Omron CX-Programmer project NewProject (CX-Programmer 9.54)

# PLC Station1: CJ1M CPU11

## Global symbols (name address type ; comment)
0.00 BOOL  ; Start_PB
0.01 BOOL  ; Stop_PB
0.02 BOOL  ; Reset_PB
0.03 BOOL  ; Emergency_PB
0.04 BOOL  ; Pusher 1 Front Limit
0.05 BOOL  ; RM Vision
0.06 BOOL  ; Diff_Sensor1
1.00 BOOL  ; RM Emitter
1.01 BOOL  ; Start_Light
1.02 BOOL  ; Stop_Light
1.03 BOOL  ; Reset_Light
1.04 BOOL  ; Pusher 1
1.05 BOOL  ; RM Roller Stopper
1.06 BOOL  ; RM Conveyor
1.07 BOOL  ; Curved RM Conveyor
1.08 BOOL  ; Check RM Conveyor
1.09 BOOL  ; Curved Reject Conveyor
1.10 BOOL  ; Reject RM Conveyor
1.11 BOOL  ; Base Machining Conveyor
D10 CHANNEL  ; Raw Metal Counting
D11 CHANNEL  ; Reject Counting
W10.00 BOOL  ; Pusher_Control
W10.01 BOOL  ; RM Roller Stopper Control
W10.02 BOOL  ; Emitter Control
W10.03 BOOL  ; Reset Counting
W1.00 BOOL  ; Status
W1.01 BOOL  ; Emergency_Status

## Program NewProgram1 (cyclic task 0)

### Section Station1

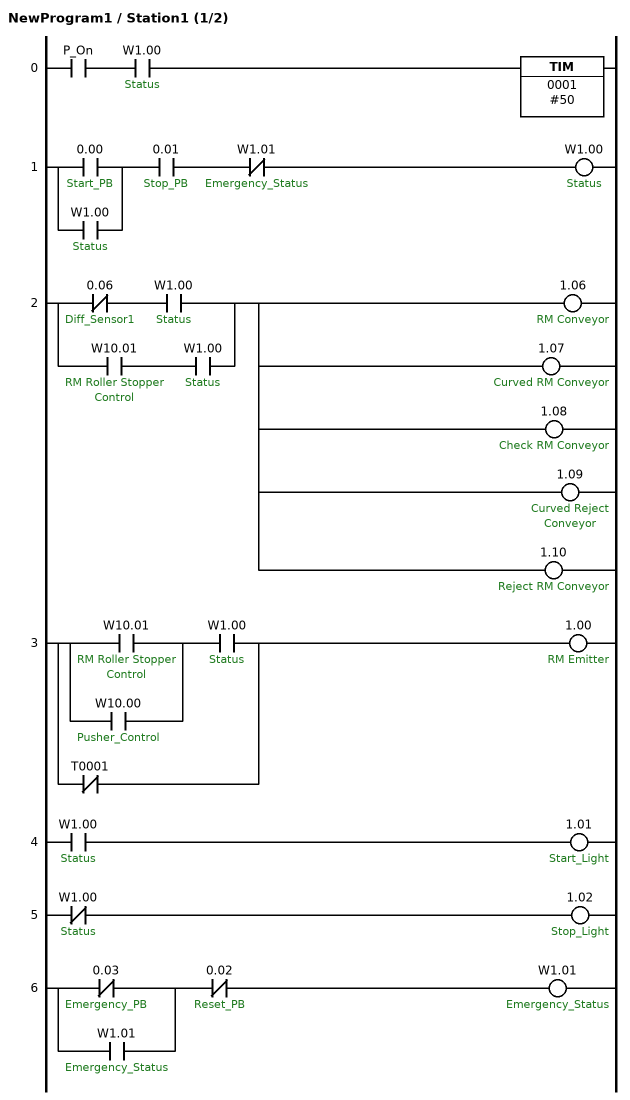
; rung 0
LD P_On
AND W1.00  ; Status
TIM 0001 #50
; rung 1
LD 0.00  ; Start_PB
OR W1.00  ; Status
AND 0.01  ; Stop_PB
ANDNOT W1.01  ; Emergency_Status
OUT W1.00  ; Status
; rung 2
LDNOT 0.06  ; Diff_Sensor1
AND W1.00  ; Status
LD W10.01  ; RM Roller Stopper Control
AND W1.00  ; Status
ORLD
OUT 1.06  ; RM Conveyor
OUT 1.07  ; Curved RM Conveyor
OUT 1.08  ; Check RM Conveyor
OUT 1.09  ; Curved Reject Conveyor
OUT 1.10  ; Reject RM Conveyor
; rung 3
LD W10.01  ; RM Roller Stopper Control
OR W10.00  ; Pusher_Control
AND W1.00  ; Status
ORNOT T0001
OUT 1.00  ; RM Emitter
; rung 4
LD W1.00  ; Status
OUT 1.01  ; Start_Light
; rung 5
LDNOT W1.00  ; Status
OUT 1.02  ; Stop_Light
; rung 6
LDNOT 0.03  ; Emergency_PB
OR W1.01  ; Emergency_Status
ANDNOT 0.02  ; Reset_PB
OUT W1.01  ; Emergency_Status

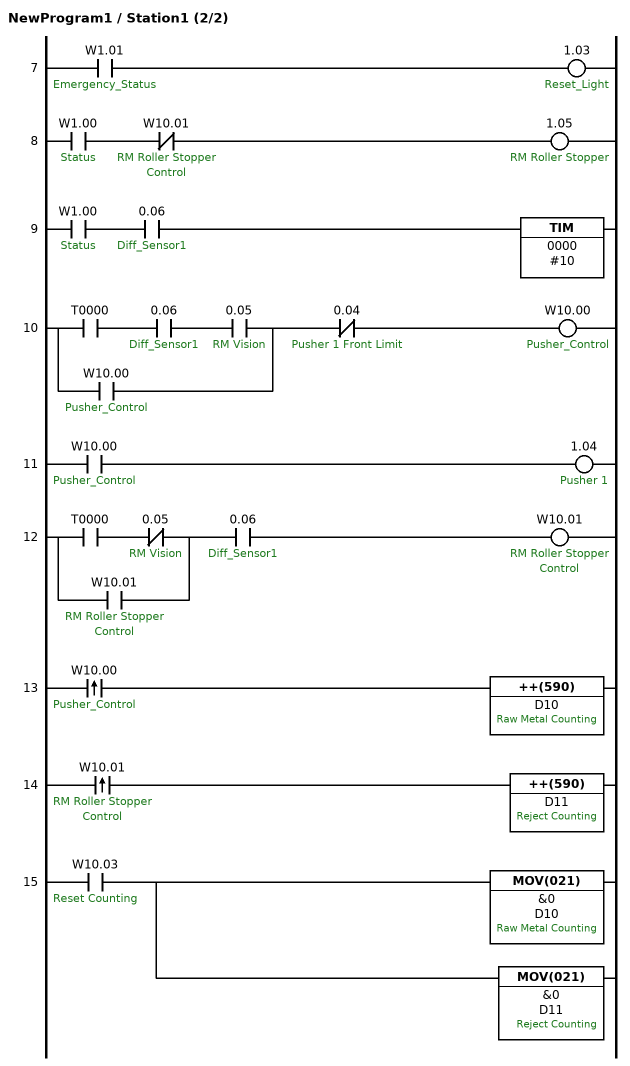
; rung 7
LD W1.01  ; Emergency_Status
OUT 1.03  ; Reset_Light
; rung 8
LD W1.00  ; Status
ANDNOT W10.01  ; RM Roller Stopper Control
OUT 1.05  ; RM Roller Stopper
; rung 9
LD W1.00  ; Status
AND 0.06  ; Diff_Sensor1
TIM 0000 #10
; rung 10
LD T0000
AND 0.06  ; Diff_Sensor1
AND 0.05  ; RM Vision
OR W10.00  ; Pusher_Control
ANDNOT 0.04  ; Pusher 1 Front Limit
OUT W10.00  ; Pusher_Control
; rung 11
LD W10.00  ; Pusher_Control
OUT 1.04  ; Pusher 1
; rung 12
LD T0000
ANDNOT 0.05  ; RM Vision
OR W10.01  ; RM Roller Stopper Control
AND 0.06  ; Diff_Sensor1
OUT W10.01  ; RM Roller Stopper Control
; rung 13
@LD W10.00  ; Pusher_Control
++(590) D10  ; Raw Metal Counting
; rung 14
@LD W10.01  ; RM Roller Stopper Control
++(590) D11  ; Reject Counting
; rung 15
LD W10.03  ; Reset Counting
MOV(021) &0 D10  ; Raw Metal Counting
MOV(021) &0 D11  ; Reject Counting

### Section HMI_Mapping

### Section END
; rung 0
END(001)